FUNCTION_BLOCK FB_Quenching
VAR_INPUT
	bExecute		: BOOL;
END_VAR
VAR_OUTPUT
	bDone			: BOOL;
	bError			: BOOL;
	wErrorID		: BOOL;
END_VAR
VAR
	
END_VAR

END_FUNCTION_BLOCK

(* stored: Version 1.1.0.1, ProductVersion 3.1.4024.11
   POU FB_Quenching: Id {ae0e565e-f920-4c0b-a44c-4def04d45a19}, SpecialFunc None *)
